(* CODESYS project Tc3_Mc3Base.library
   TcLibraryId: Beckhoff Automation GmbH|Tc3_Mc3Base|0.4.47.0
   Company: Beckhoff Automation GmbH
   Title: Tc3_Mc3Base
   Placeholder: Tc3_Mc3Base
   Version: 0.4.47.0

Project tree, tasks and I/O mapping:
  POUs/
    TestCommands/
      function block MC_ForceObjectError [ST]: FB_init, FB_exit
      function block MC_NotSupportedCommand [ST]: FB_init, FB_exit
      function block MC_FailProcessCommand [ST]: FB_init, FB_exit
  DUTs/
    Enums/
      data type EBufferMode
      data type ESyncDirection
      data type ESyncStrategy
      data type EPositionInterpretation
      data type ESignalEdgeEvaluation
      data type EReactionToMasterError
      data type EReactionToSlaveError
    Structs/
      data type DriveInfo
    interface Type_MotionObject: GetMotionObjectOid
  Version/
    global variables Global_Version
*)

// DUTs/Enums/EBufferMode
(* Buffer mode between buffered commands. *)
{attribute 'TcIecLibraryType'}
{attribute 'Namespace' := 'Tc3_Mc3Base'}
{attribute 'qualified_only'}
{attribute 'strict'}
{attribute 'to_string'}
TYPE EBufferMode : (
	Aborting:=0, 	(* The previous command is aborted and a transition to the new command is initiated immediately. *)
	Buffered:=1, 	(* The previous command is executed to completion. The new command affects the motion object as 
		soon as the previous movement is 'Done'/'InVelocity'/'InSync'/'InGear'. There is no blending. *)
	BlendingLow:=18	(* The new command is executed as soon as the motion object is no longer executing any other command. Unlike Buffered, the motion object 
		does not stop at the previous target position, but instead moves through this position at the lower speed of two commands. *)
) UINT;
END_TYPE

// DUTs/Enums/ESyncDirection
(* Directions in which a slave is allowed to move during synchronizing phase. *)
{attribute 'TcIecLibraryType'}
{attribute 'Namespace' := 'Tc3_Mc3Base'}
{attribute 'qualified_only'}
{attribute 'strict'}
{attribute 'to_string'}
TYPE ESyncDirection : (
		{attribute 'hide'}
Invalid:=0, 	(* Indicates invalid information, e.g. no connection or component not yet ready. *)
	Positive:=1, 	(* Movement is allowed only in positive direction while synchronizing. *)
	Negative:=2, 	(* Movement is allowed only in negative direction while synchronizing. *)
	Both:=3	(* Movement is allowed in any direction while synchronizing. *)
) UINT := Invalid;
END_TYPE

// DUTs/Enums/ESyncStrategy
{attribute 'TcIecLibraryType'}
{attribute 'Namespace' := 'Tc3_Mc3Base'}
{attribute 'qualified_only'}
{attribute 'strict'}
{attribute 'to_string'}
TYPE ESyncStrategy : (Late:=1, Slow:=2, Early:=3) UINT;
END_TYPE

// DUTs/Enums/EPositionInterpretation
(* Interpretation of position as modulo or absolute. *)
{attribute 'TcIecLibraryType'}
{attribute 'Namespace' := 'Tc3_Mc3Base'}
{attribute 'qualified_only'}
{attribute 'strict'}
{attribute 'to_string'}
TYPE EPositionInterpretation : (
	Absolute:=0, 	(* Position is interpreted as an absolute value. *)
	ModuloPositiveDirection:=1, 	(* Position is interpreted as a modulo value. The direction of movement 
		is positive direction. *)
	ModuloShortestDistance:=2, 	(* Position is interpreted as a modulo value. The direction of movement depends 
		on whether the shortest distance to the target position is determined by the positive direction 
		of movement or the negative direction of movement. *)
	ModuloNegativeDirection:=3	(* Position is interpreted as a modulo value. The direction of movement 
		is negative direction. *)
) UINT;
END_TYPE

// DUTs/Enums/ESignalEdgeEvaluation
(* Specifies which signal change or rather which signal edge is decisive. *)
{attribute 'TcIecLibraryType'}
{attribute 'Namespace' := 'Tc3_Mc3Base'}
{attribute 'qualified_only'}
{attribute 'strict'}
{attribute 'to_string'}
TYPE ESignalEdgeEvaluation : (
	RisingEdge:=0, 	(* Rising signal edge is decisive. *)
	FallingEdge:=1	(* Falling signal edge is decisive. *)
) UINT;
END_TYPE

// DUTs/Enums/EReactionToMasterError
(* Reaction type to master errors in master/slave couplings. *)
{attribute 'TcIecLibraryType'}
{attribute 'Namespace' := 'Tc3_Mc3Base'}
{attribute 'qualified_only'}
{attribute 'strict'}
{attribute 'to_string'}
TYPE EReactionToMasterError : (
	TriggerSlaveError:=0, 	(* In case of a master error a slave error is triggered. *)
	KeepCouplingWithSetValues:=1	(* In case of a master error the coupling is kept with set values and no 
		slave error is triggered. *)
) UINT;
END_TYPE

// DUTs/Enums/EReactionToSlaveError
(* Reaction type to slave errors in master/slave couplings. *)
{attribute 'TcIecLibraryType'}
{attribute 'Namespace' := 'Tc3_Mc3Base'}
{attribute 'qualified_only'}
{attribute 'strict'}
{attribute 'to_string'}
TYPE EReactionToSlaveError : (
	TriggerMasterError:=0, 	(* In case of a slave error a master error is triggered. *)
	NoReaction:=1	(* No reaction on the master in case of a slave error. *)
) UINT;
END_TYPE

// DUTs/Structs/DriveInfo
{attribute 'TcIecLibraryType'}
{attribute 'Namespace' := 'Tc3_Mc3Base'}
TYPE DriveInfo : 
	STRUCT
		(* Drive netId and port *)
		{attribute 'GUID' := '18071995-0000-0000-0000-000000000042'}
		AmsAddress : GLOBAL.AMSADDR;
		(* Drive Channel Number *)
		ChannelNumber : DINT;
	END_STRUCT
END_TYPE

// Version/Global_Version
{attribute 'TcGenerated'}
// This function has been automatically generated from the project information.
VAR_GLOBAL CONSTANT
	{attribute 'const_non_replaced'}
	{attribute 'linkalways'}
	stLibVersion_Tc3_Mc3Base : ST_LibVersion := (iMajor := 0, iMinor := 4, iBuild := 47, iRevision := 0, nFlags := 0, sVersion := '0.4.47.0');
	{attribute 'const_non_replaced'}
	{attribute 'linkalways'}
	sLibraryId_Tc3_Mc3Base : String := 'Beckhoff Automation GmbH|Tc3_Mc3Base|0.4.47.0';
END_VAR

// DUTs/Type_MotionObject
{attribute 'Namespace' := 'Tc3_Mc3Base'}
{attribute 'c++_compatible'}
INTERFACE Type_MotionObject

{attribute 'TcTypeSystem'}
{attribute 'c++_compatible'}
{attribute 'minimal_input_size' := '4'}
{attribute 'pack_mode' := '4'}
{attribute 'hide'}
METHOD GetMotionObjectOid : GLOBAL.OTCID
END_METHOD

END_INTERFACE

// POUs/TestCommands/MC_ForceObjectError

{attribute 'c++_compatible'}
{attribute 'external_name' := 'MC_ForceObjectError_GUID_2C21623D_7607_A703_3DAD_6F12C443FC2C'}
{attribute 'TcIecLibraryType'}
{attribute 'hide_all_locals'}
(* 
		This function block commands an axis error.
	 *)
FUNCTION_BLOCK MC_ForceObjectError
VAR_INPUT
	(* Object Id of the object on which the error should be enforced (e.g. Axis Oid, LinearMover Oid, Group Oid). *)
	{attribute 'GUID' := '18071995-0000-0000-0000-00000000000F'}
	{attribute 'GlobalType'}
	Oid : GLOBAL.OTCID;
	(* Trigger the command with rising edge *)
	Execute : BOOL;
END_VAR
VAR
	 {attribute 'hide'}
	_reserved1 : ARRAY [1..3] OF USINT;
END_VAR
VAR_INPUT
	(* Error code to be triggered *)
	ErrorCode : UDINT;
	ControlError : BOOL;
END_VAR
VAR_OUTPUT
	(* Error has been successfully triggered *)
	Done : BOOL;
	(* Function block is not finished and new output values are to be expected *)
	Busy : BOOL;
	(* Error occurred within function block *)
	Error : BOOL;
	(* Error identifier *)
	ErrorId : UDINT;
END_VAR
VAR
	 {attribute 'hide'}
	_reserved2 : UINT_0_32;
	 {attribute 'hide'}
	_reserved3 : ARRAY [1..40] OF UINT_8_16;
	 {attribute 'hide'}
	_reserved4 : ARRAY [1..8] OF USINT;
END_VAR

{attribute 'TcTypeSystem'}

(* Internal method *)
{attribute 'hide'}
METHOD FB_init : BOOL
VAR_INPUT
	(*  if TRUE, the retain variables are initialized (warm start / cold start) *)
	bInitRetains : BOOL;
	(*  if TRUE, the instance afterwards gets moved into the copy code (online change) *)
	bInCopyCode : BOOL;
END_VAR
END_METHOD

{attribute 'TcTypeSystem'}

(* Internal method *)
{attribute 'hide'}
METHOD FB_exit : BOOL
VAR_INPUT
	(*  if TRUE, the exit method is called for exiting an instance that is copied afterwards (online change). *)
	bInCopyCode : BOOL;
END_VAR
END_METHOD

END_FUNCTION_BLOCK

// POUs/TestCommands/MC_NotSupportedCommand

{attribute 'c++_compatible'}
{attribute 'external_name' := 'MC_NotSupportedCommand_GUID_EEC71BDE_BD37_AE21_325D_9CB6C3E209E4'}
{attribute 'TcIecLibraryType'}
{attribute 'hide'}
{attribute 'hide_all_locals'}
FUNCTION_BLOCK MC_NotSupportedCommand
VAR_INPUT
	(* Object Id of the object to which this command is sent (e.g. Axis Oid, LinearMover Oid, Group Oid) *)
	{attribute 'GUID' := '18071995-0000-0000-0000-00000000000F'}
	{attribute 'GlobalType'}
	Oid : GLOBAL.OTCID;
	(* Trigger the command with rising edge *)
	Execute : BOOL;
END_VAR
VAR
	 {attribute 'hide'}
	_reserved1 : ARRAY [1..3] OF USINT;
END_VAR
VAR_INPUT
	FailIn : UDINT;
END_VAR
VAR_OUTPUT
	(* Indicates if the command has been executed successfully *)
	Done : BOOL;
	(* Function block is not finished and new output values are to be expected *)
	Busy : BOOL;
	(* Function block has active control on the axis *)
	Active : BOOL;
	(* Command is aborted by another command *)
	CommandAborted : BOOL;
	(* Error occurred within function block *)
	Error : BOOL;
END_VAR
VAR
	 {attribute 'hide'}
	_reserved2 : ARRAY [1..3] OF USINT;
END_VAR
VAR_OUTPUT
	(* Error identifier *)
	ErrorId : UDINT;
END_VAR
VAR
	 {attribute 'hide'}
	_reserved3 : UINT_0_32;
	 {attribute 'hide'}
	_reserved4 : ARRAY [1..36] OF UINT_8_16;
	 {attribute 'hide'}
	_reserved5 : ARRAY [1..12] OF USINT;
END_VAR

{attribute 'TcTypeSystem'}

(* Internal method *)
{attribute 'hide'}
METHOD FB_init : BOOL
VAR_INPUT
	(*  if TRUE, the retain variables are initialized (warm start / cold start) *)
	bInitRetains : BOOL;
	(*  if TRUE, the instance afterwards gets moved into the copy code (online change) *)
	bInCopyCode : BOOL;
END_VAR
END_METHOD

{attribute 'TcTypeSystem'}

(* Internal method *)
{attribute 'hide'}
METHOD FB_exit : BOOL
VAR_INPUT
	(*  if TRUE, the exit method is called for exiting an instance that is copied afterwards (online change). *)
	bInCopyCode : BOOL;
END_VAR
END_METHOD

END_FUNCTION_BLOCK

// POUs/TestCommands/MC_FailProcessCommand

{attribute 'c++_compatible'}
{attribute 'external_name' := 'MC_FailProcessCommand_GUID_E9BBDF78_8DFF_A075_39BB_D4A139F2834E'}
{attribute 'TcIecLibraryType'}
{attribute 'hide'}
{attribute 'hide_all_locals'}
(* 
		This function block commands an axis error.
	 *)
FUNCTION_BLOCK MC_FailProcessCommand
VAR_INPUT
	(* Object Id of the object that receives this command (e.g. Axis Oid, LinearMover Oid, Group Oid) *)
	{attribute 'GUID' := '18071995-0000-0000-0000-00000000000F'}
	{attribute 'GlobalType'}
	Oid : GLOBAL.OTCID;
	(* Trigger the command with rising edge *)
	Execute : BOOL;
END_VAR
VAR_OUTPUT
	(* Error has been successfully triggered *)
	Done : BOOL;
	(* Function block is not finished and new output values are to be expected *)
	Busy : BOOL;
	(* Function block has active control on the axis *)
	Active : BOOL;
	(* Command is aborted by another command *)
	CommandAborted : BOOL;
	(* Error occurred within function block *)
	Error : BOOL;
END_VAR
VAR
	 {attribute 'hide'}
	_reserved1 : UINT;
END_VAR
VAR_OUTPUT
	(* Error identifier *)
	ErrorId : UDINT;
END_VAR
VAR
	 {attribute 'hide'}
	_reserved2 : UINT_0_32;
	 {attribute 'hide'}
	_reserved3 : ARRAY [1..36] OF UINT_8_16;
	 {attribute 'hide'}
	_reserved4 : ARRAY [1..12] OF USINT;
END_VAR

{attribute 'TcTypeSystem'}

(* Internal method *)
{attribute 'hide'}
METHOD FB_init : BOOL
VAR_INPUT
	(*  if TRUE, the retain variables are initialized (warm start / cold start) *)
	bInitRetains : BOOL;
	(*  if TRUE, the instance afterwards gets moved into the copy code (online change) *)
	bInCopyCode : BOOL;
END_VAR
END_METHOD

{attribute 'TcTypeSystem'}

(* Internal method *)
{attribute 'hide'}
METHOD FB_exit : BOOL
VAR_INPUT
	(*  if TRUE, the exit method is called for exiting an instance that is copied afterwards (online change). *)
	bInCopyCode : BOOL;
END_VAR
END_METHOD

END_FUNCTION_BLOCK
